Staubli VAL3: processList.dtx

num nFile
string sEvent
string sProcessList
string sType
string sWrite
bool bLoading
public bool bLoop = true
